(* Logix 5000 project; controller HotdogAb 1769-L16ER-BB1B rev 32.11; software revision 32.00 *)

TASK MainTask (continuous, watchdog 500 ms) : Hotdog

MODULES
   Local : 1769-L16ER-BB1B (PointIO 0, rev 32.11)
      Discrete_IO : Embedded (PointIO 1, rev 32.11, Output RPI 20 ms)
END_MODULES

VAR_GLOBAL   (* controller tags *)
   count_up : COUNTER;
   hotdog : BOOL;
   ketchup_remem : BOOL;
   mustard_remem : BOOL;
END_VAR

PROGRAM Hotdog   (* main routine MainRoutine *)
VAR
   ketchup : BOOL;
   mustard : BOOL;
END_VAR

ROUTINE MainRoutine   (* ladder *)
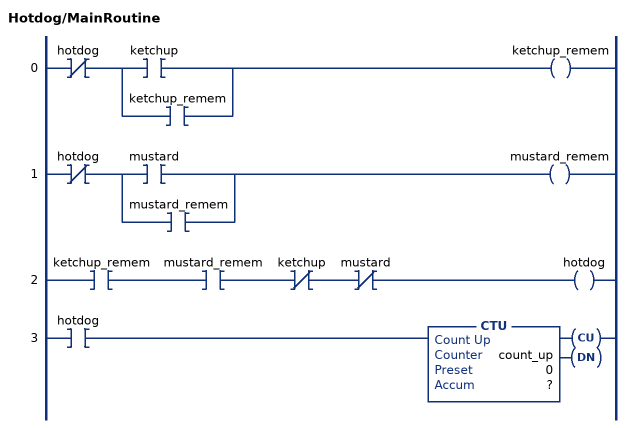
   0: XIO(hotdog)[XIC(ketchup) ,XIC(ketchup_remem) ]OTE(ketchup_remem);
   1: XIO(hotdog)[XIC(mustard) ,XIC(mustard_remem) ]OTE(mustard_remem);
   2: XIC(ketchup_remem)XIC(mustard_remem)XIO(ketchup)XIO(mustard)OTE(hotdog);
   3: XIC(hotdog)CTU(count_up,?,?);
END_ROUTINE
END_PROGRAM
